PROGRAM MAIN
VAR
    axis: AXIS_REF;
	MC_ReadActualPosition: MC_ReadActualPosition;
	MC_ReadActualVelocity: MC_ReadActualVelocity;
	state: state;
	
	reset_output:ST_McOutputs;
	axis_Reset: MC_Reset;
	ReadP_Valid:BOOL;
	ReadV_Valid:BOOL;
	Position: LREAL;
	Velocity: LREAL;
	power1: MC_Power;
	power1_output:ST_McOutputs;
END_VAR

// Programmablauf mittels Zustandsautomat
CASE state OF
	
	INIT:
		GVL.MC_MoveAbsolute.Execute := FALSE;
		Power1.Enable:=FALSE;
		axis_Reset.Execute:=FALSE;
		state := POWER_ON;
	
	POWER_ON:
		Power1.Enable := TRUE;
		IF power1_output.Done = TRUE THEN
			state := MOVE_ON;
		ELSIF power1_output.Done = FALSE THEN
			state := POWER_ON;
		END_IF
		IF axis.Status.Error THEN
			state := ERROR;
		END_IF
 
	MOVE_ON:
		IF GVL.MC_MoveAbsolute_output.Busy = FALSE THEN	
			GVL.MC_MoveAbsolute.Velocity := 10;
			GVL.MC_MoveAbsolute.Execute := TRUE;
			//state := MOVE_ON;
		END_IF
		
		IF GVL.MC_MoveAbsolute.Done THEN
			state := INIT;
		END_IF
		
		IF axis.Status.Error THEN
			state := ERROR;
		END_IF
		
	ERROR:
		GVL.MC_MoveAbsolute.Execute:=FALSE;
		IF NOT axis.Status.Coupled THEN
			IF axis.Status.Error THEN
				state := P_RESET;	
			ELSE
				state := INIT;
			END_IF
		END_IF
		
	P_RESET:
		axis_Reset.Execute := TRUE;
		GVL.MC_MoveAbsolute.Execute:=FALSE;
			
			IF axis_Reset.Done  THEN
				state := INIT;
			ELSIF axis_Reset.Error  THEN
				state := INIT; 
			END_IF
END_CASE

axis();
Signalersteller();
power();
MoveAbsolute();
ReadP_V();
reset();

ACTION MoveAbsolute:
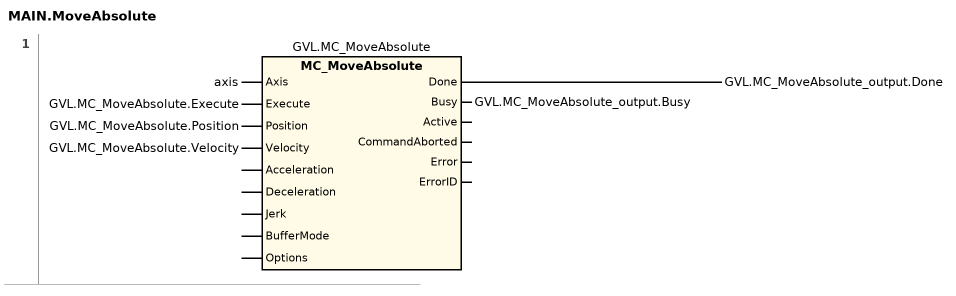
// NETWORK 1
GVL.MC_MoveAbsolute(
    Axis := axis,
    Execute := GVL.MC_MoveAbsolute.Execute,
    Position := GVL.MC_MoveAbsolute.Position,
    Velocity := GVL.MC_MoveAbsolute.Velocity,
    Busy => GVL.MC_MoveAbsolute_output.Busy); // MC_MoveAbsolute
GVL.MC_MoveAbsolute_output.Done := GVL.MC_MoveAbsolute.Done;
END_ACTION

ACTION PID:
// NETWORK 1
END_ACTION

ACTION Power:
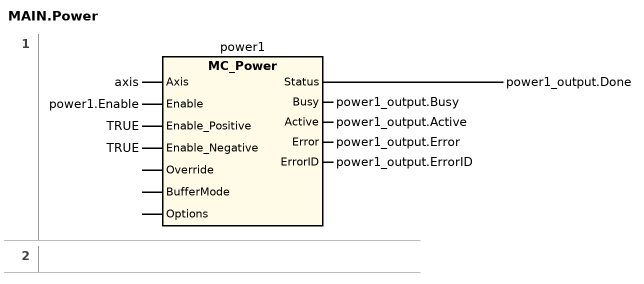
// NETWORK 1
power1(
    Axis := axis,
    Enable := power1.Enable,
    Enable_Positive := TRUE,
    Enable_Negative := TRUE,
    Busy => power1_output.Busy,
    Active => power1_output.Active,
    Error => power1_output.Error,
    ErrorID => power1_output.ErrorID); // MC_Power
power1_output.Done := power1.Status;

// NETWORK 2
END_ACTION

ACTION ReadP_V:
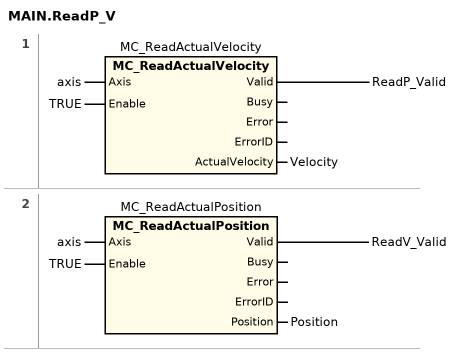
// NETWORK 1
MC_ReadActualVelocity(Axis := axis, Enable := TRUE, ActualVelocity => Velocity);
ReadP_Valid := MC_ReadActualVelocity.Valid;

// NETWORK 2
MC_ReadActualPosition(Axis := axis, Enable := TRUE, Position => Position);
ReadV_Valid := MC_ReadActualPosition.Valid;
END_ACTION

ACTION Reset:
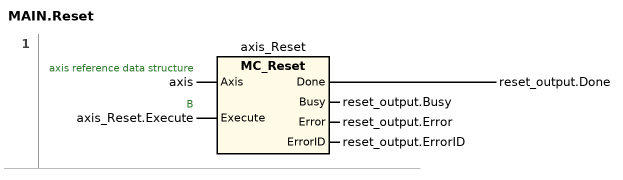
// NETWORK 1
//   axis: axis reference data structure
//   axis_Reset.Execute: B
axis_Reset(
    Axis := axis,
    Execute := axis_Reset.Execute,
    Busy => reset_output.Busy,
    Error => reset_output.Error,
    ErrorID => reset_output.ErrorID); // MC_Reset
reset_output.Done := axis_Reset.Done;
END_ACTION

END_PROGRAM

(* stored: Version 1.1.0.1, ProductVersion 3.1.4024.9
   POU MAIN: Id {534445fb-a9af-45c0-84b6-2e30f7c91eb2}, SpecialFunc None
   Action MoveAbsolute: Id {4da0892b-5491-4bc8-980a-fbafe0d598e8}
   Action PID: Id {f0f4cc91-567b-4677-9454-8daa0a88b5d5}
   Action Power: Id {8b469144-5c09-487e-8637-7d166d37593e}
   Action ReadP_V: Id {4fb1b366-fac7-45a0-822a-d6e5a92b9fcd}
   Action Reset: Id {d4c531c5-ab2c-485e-947c-8ec7bbf86e8a} *)
